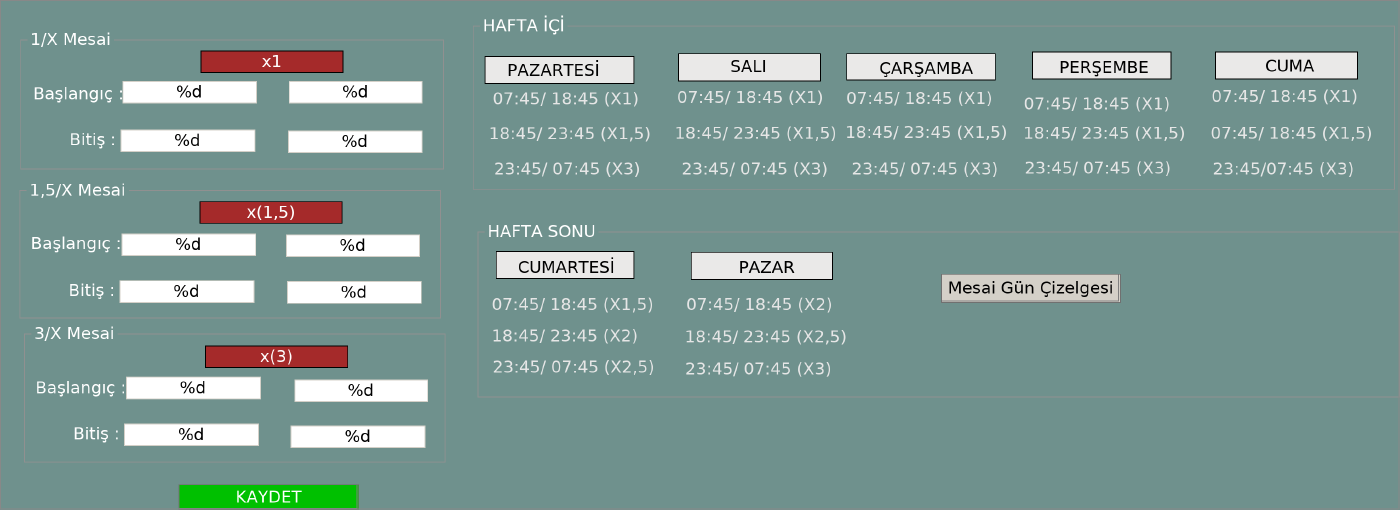
VISUALIZATION MesaiSaat_sayfa  // 1522x555
    Button (194,527 196x28), "KAYDET"
        toggle GVL_mesai_saat.kaydet
        OnMouseClick: change screen: Hesap_Sayfa
    Button (1023,298 195x31), "Mesai Gün Çizelgesi"
        OnMouseClick: change screen: gun_cizelge
    GroupBox (514,20 1002x186), "HAFTA İÇİ"
        Rectangle (807,36 155x30)
        Rectangle (608,36 151x30)
        Rectangle (406,38 162x29)
        Rectangle (223,38 155x30)
        Rectangle (13,41 162x30)
        Label (10,36 156x41), "PAZARTESİ"
        Label (227,28 146x49), "SALI"
        Label (414,32 159x45), "ÇARŞAMBA"
        Label (616,36 141x35), "PERŞEMBE"
        Label (818,30 141x44), "CUMA"
        Label (21,63 160x49), "07:45/ 18:45 (X1)"
        Label (21,101 169x49), "18:45/ 23:45 (X1,5)"
        Label (15,81 169x30)
        Label (217,71 169x30), "07:45/ 18:45 (X1)"
        Label (223,102 169x46), "18:45/ 23:45 (X1,5)"
        Label (401,72 169x30), "07:45/ 18:45 (X1)"
        Label (406,109 174x30), "18:45/ 23:45 (X1,5)"
        Label (594,78 169x30), "07:45/ 18:45 (X1)"
        Label (595,110 183x30), "18:45/ 23:45 (X1,5)"
        Label (798,70 169x30), "07:45/ 18:45 (X1)"
        Label (802,110 176x30), "07:45/ 18:45 (X1,5)"
        Label (797,149 169x30), "23:45/07:45 (X3)"
        Label (595,148 169x30), "23:45/ 07:45 (X3)"
        Label (407,149 169x30), "23:45/ 07:45 (X3)"
        Label (222,149 169x30), "23:45/ 07:45 (X3)"
        Label (18,149 169x30), "23:45/ 07:45 (X3)"
    GroupBox (519,244 1003x188), "HAFTA SONU"
        Rectangle (20,29 150x30)
        Label (20,32 154x30), "CUMARTESİ"
        Rectangle (232,30 154x30)
        Label (231,28 167x38), "PAZAR"
        Label (16,63 175x49), "07:45/ 18:45 (X1,5)"
        Label (15,98 160x47), "18:45/ 23:45 (X2)"
        Label (219,63 175x49), "07:45/ 18:45 (X2)"
        Label (228,98 171x49), "18:45/ 23:45 (X2,5)"
        Label (212,133 187x49), "23:45/ 07:45 (X3)"
    Label (535,375 177x49), "23:45/ 07:45 (X2,5)"
    GroupBox (22,35 460x149), "1/X Mesai"
        Textfield (111,53 146x24), "%d", text variable: GVL_mesai_saat.x1bslangicSaat
            OnMouseClick: write the text variable via VisuDialogs.Numpad, min 8, max 19
        Textfield (292,53 145x24), "%d", text variable: GVL_mesai_saat.x1bslangicdakika
            OnMouseClick: write the text variable via VisuDialogs.Numpad, min 0, max 59
        Textfield (109,106 146x24), "%d", text variable: GVL_mesai_saat.x1bitisSaat
            OnMouseClick: write the text variable via VisuDialogs.Numpad, min 8, max 19
        Textfield (291,107 146x24), "%d", text variable: GVL_mesai_saat.x1bitisdakika
            OnMouseClick: write the text variable via VisuDialogs.Numpad, min 0, max 59
        Rectangle (196,20 155x24), "x1"
        Label (4,102 150x30), "Bitiş :"
    Label (14,87 143x30), "Başlangıç :"
    GroupBox (21,199 458x147), "1,5/X Mesai"
        Textfield (111,55 146x24), "%d", text variable: GVL_mesai_saat.x1_5bslangicSaat
            OnMouseClick: write the text variable via VisuDialogs.Numpad, min 19, max 23
        Textfield (290,56 145x24), "%d", text variable: GVL_mesai_saat.x1_5bslangicdakika
            OnMouseClick: write the text variable via VisuDialogs.Numpad, min 0, max 59
        Textfield (109,106 146x24), "%d", text variable: GVL_mesai_saat.x1_5bitisSaat
            OnMouseClick: write the text variable via VisuDialogs.Numpad, min 19, max 23
        Textfield (291,107 146x24), "%d", text variable: GVL_mesai_saat.x1_5bitisdakika
            OnMouseClick: write the text variable via VisuDialogs.Numpad, min 0, max 59
        Label (4,102 150x30), "Bitiş :"
        Rectangle (196,20 155x24), "x(1,5)"
    Label (8,250 150x30), "Başlangıç :"
    GroupBox (26,355 458x148), "3/X Mesai"
        Textfield (111,55 146x24), "%d", text variable: GVL_mesai_saat.x3bslangicSaat
            OnMouseClick: write the text variable via VisuDialogs.Numpad
        Textfield (294,58 145x24), "%d", text variable: GVL_mesai_saat.x3bslangicdakika
            OnMouseClick: write the text variable via VisuDialogs.Numpad, min 45
        Textfield (109,106 146x24), "%d", text variable: GVL_mesai_saat.x3bitisSaat
            OnMouseClick: write the text variable via VisuDialogs.Numpad
        Textfield (290,108 146x24), "%d", text variable: GVL_mesai_saat.x3bitisdakika
            OnMouseClick: write the text variable via VisuDialogs.Numpad
        Label (4,102 150x30), "Bitiş :"
        Rectangle (197,21 155x24), "x(3)"
    Label (13,407 150x30), "Başlangıç :"
END_VISUALIZATION

(* stored: Version 1.1.0.1, ProductVersion 3.1.4024.12
   Visu MesaiSaat_sayfa: Id {422a43d6-51dd-4fd2-9af5-5cffda930cbf} *)
